// TIA Portal V20 export
// export: Created 2025-12-01T14:56:18.0884461Z, ExportSetting None, DisplayName Totally Integrated Automation Portal, DisplayVersion V20 Update 3, DisplayName TIA Portal Openness, DisplayVersion V20 Update 3, DisplayName TIA Portal Version Control Interface, DisplayVersion V20 Update 3, DisplayName STEP 7 Professional, DisplayVersion V20 Update 3, DisplayName STEP 7 Safety, DisplayVersion V20 Update 2, DisplayName WinCC Basic/Comfort/Advanced, DisplayVersion V20 Update 3, DisplayName WinCC Professional, DisplayVersion V20 Update 3, DisplayName WinCC Unified, DisplayVersion V20 Update 3
TYPE "Status_Word_MX2_V2"
   STRUCT
      Frequecy_Arrival : Bool;   // (FA)Frequency Arrival (Frecuencia alcanzada) =1
      Control_Status : Bool;   // (CS)Control Status =1 Profibus in control
      Reservado_bit_10 : Bool;   // siempre a 0
      Reservado_bit_11 : Bool;   // siempre a 0
      Reservado_bit_12 : Bool;   // siempre a 0
      Reservado_bit_13 : Bool;   // siempre a 0
      Reservado_bit_14 : Bool;   // siempre a 0
      Reservado_bit_15 : Bool;   // siempre a 0
      Reservado_bit_0 : Bool;   // siempre a 1
      AC_Mains : Bool;   // AC Main on =1;AC Main off =0 (tensión principal)
      Ready : Bool;   // (Rdy) =1 Variador preparado
      Fault : Bool;   // (Flt) = 1 en fallo
      Reservado_bit_4 : Bool;   // siempre a 1
      Reservado_bit_5 : Bool;   // siempre a 1
      Reservado_bit_6 : Bool;   // siempre a 0
      Alarm : Bool;   // (Alm) = 1 en alarma
   END_STRUCT;
END_TYPE
